ABB RAPID module: 00369D41

MODULE PickUpDownBlock

    PROC Temp()
        PickBlock 0, 407, 157, [0, 0, -1, 0];    ENDPROC


    PROC PickBlock(num X, num Y, num Z, orient Quat)
        VAR robtarget AboveBlock;
        VAR robtarget OnBlock;
        AboveBlock := pTableHome;
        OnBlock := pTableHome;

        AboveBlock.trans := [X, Y, 170];
        AboveBlock.rot := Quat;
        OnBlock.trans := [X, Y, Z];
        OnBlock.rot := Quat;

        MoveJ AboveBlock, defaultSpeed, fine, tSCup;
        MoveJ OnBlock, defaultSpeed, fine, tSCup;

        WaitTime 0.5;
        TurnVacOn;
        WaitTime 0.5;

        MoveJ AboveBlock, defaultSpeed, fine, tSCup;

    ENDPROC

    PROC DropBlock(num X, num Y, num Z, orient Quat)
        VAR robtarget AboveBlock;
        VAR robtarget OnBlock;
        AboveBlock := pTableHome;
        OnBlock := pTableHome;

        AboveBlock.trans := [X, Y, 170];
        AboveBlock.rot := Quat;
        OnBlock.trans := [X, Y, Z];
        OnBlock.rot := Quat;

        MoveJ AboveBlock, defaultSpeed, fine, tSCup;
        MoveJ OnBlock, defaultSpeed, fine, tSCup;

        WaitTime 0.5;
        TurnVacOff;
        WaitTime 0.5;
        MoveJ AboveBlock, defaultSpeed, fine, tSCup;

    ENDPROC

    PROC TurnVacOn()

        ! Set Vacuum system on.
        SetDO DO10_1, 1;

        ! Set suction on
        SetDO DO10_2, 1;

    ENDPROC

    ! This function sets output 1/Vac to 0
    PROC TurnVacOff()

        ! Set suction off
        SetDO DO10_2, 0;
        ! Set Vacuum system off.
        SetDO DO10_1, 0;
    ENDPROC



ENDMODULE
